// TIA Portal V21 export
TYPE "lubricationSystemInterface"
   STRUCT
      cmd { ExternalAccessible := 'False'; ExternalVisible := 'False'; ExternalWritable := 'False'} : "lubricationSystemCmd";
      sta { ExternalAccessible := 'False'; ExternalVisible := 'False'; ExternalWritable := 'False'} : "lubricationSystemSta";
      out { ExternalAccessible := 'False'; ExternalVisible := 'False'; ExternalWritable := 'False'; S7_SetPoint := 'True'} : "lubricationSystemOut";
   END_STRUCT;
END_TYPE
